// TIA Portal V21 export
VAR_GLOBAL   // PLC tag table "KAllPid"
END_VAR
VAR_GLOBAL CONSTANT   // user constants
   KAllPid_Min_SetPoint : Int := 1;   // Mindestsollwert erreicht / Minimum setpoint reached / Alcanzado el punto de ajuste mínimo / Le point de consigne minimum atteint / Raggiunto il minimo setpoint
   KAllPid_Max_SetPoint : Int := 2;   // Maximaler sollwert erreicht / Maximum setpoint reached / Se ha alcanzado el punto de ajuste máximo / Atteint le point de consigne maximal / Raggiunto il massimo setpoint
   KAllPid_Troppo_Tempo_Allarme : Int := 3;   // Zu lange im alarmzustand / Too much time on alarm / Demasiado tiempo en alarma / Trop de temps en alarme / Troppo tempo in allarme
END_VAR
